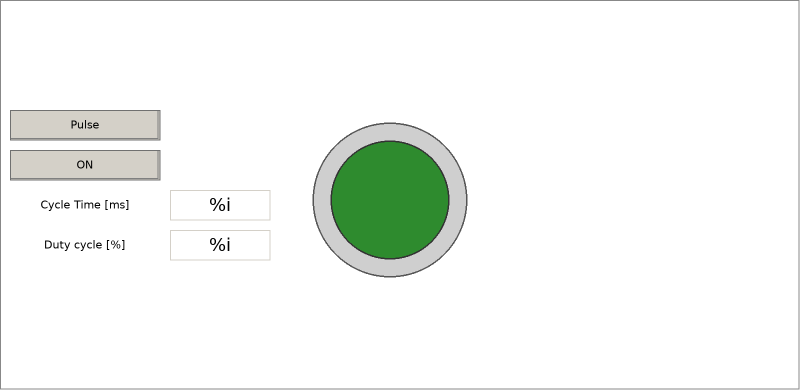
VISUALIZATION VisuPWMControl  // 800x390
VAR_IN_OUT
	fbManualControler	: FB_ManualController ;
END_VAR
    Lamp1 (300,110 180x180), variable: fbManualControler.pDevPWMController^.qbOutput, style: Lamp-Lamp1-Green
    Button (10,110 150x30), "Pulse"
        toggle fbManualControler.pDevPWMController^.bCmdPWMCycle
    Button (10,150 150x30), "ON"
        tap fbManualControler.pDevPWMController^.bCmdOn
    Textfield (170,190 100x30), "%i", text variable: fbManualControler.pDevPWMController^.nPeriodLength
        OnMouseUp: write the text variable via VisuDialogs.Numpad
    Label (10,190 150x30), "Cycle Time [ms]"
    Label (10,230 150x30), "Duty cycle [%]"
    Textfield (170,230 100x30), "%i", text variable: fbManualControler.pDevPWMController^.nDutyCycle
        OnMouseClick: write the text variable via VisuDialogs.Numpad, min 0, max 100
END_VISUALIZATION

(* stored: Version 1.1.0.1, ProductVersion 3.1.4024.9
   Visu VisuPWMControl: Id {34378a83-c52f-4e83-a907-461e917d0c7e} *)
